SUBAPPLICATION SRV_SERVER (* ROS 2 SRV Server *)
  (* Standard: 61499-2 *)
  (* Version 1.0, 2023-03-14, derPi *)
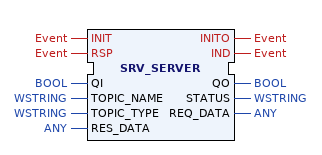
  EVENT_INPUT
    INIT; (* Initialization Request *)
    RSP; (* Application Response to IND *)
  END_EVENT
  EVENT_OUTPUT
    INITO; (* Initialization Confirm *)
    IND; (* Confirmation of Requested Service *)
  END_EVENT
  VAR_INPUT
    QI : BOOL; (* Input Event Qualifier *)
    TOPIC_NAME : WSTRING; (* ROS 2 Topic Name *)
    TOPIC_TYPE : WSTRING; (* ROS 2 Topic Type *)
    RES_DATA : ANY; (* Response Data *)
  END_VAR
  VAR_OUTPUT
    QO : BOOL; (* Output Event Qualifier *)
    STATUS : WSTRING; (* Service Status *)
    REQ_DATA : ANY; (* Request Data *)
  END_VAR
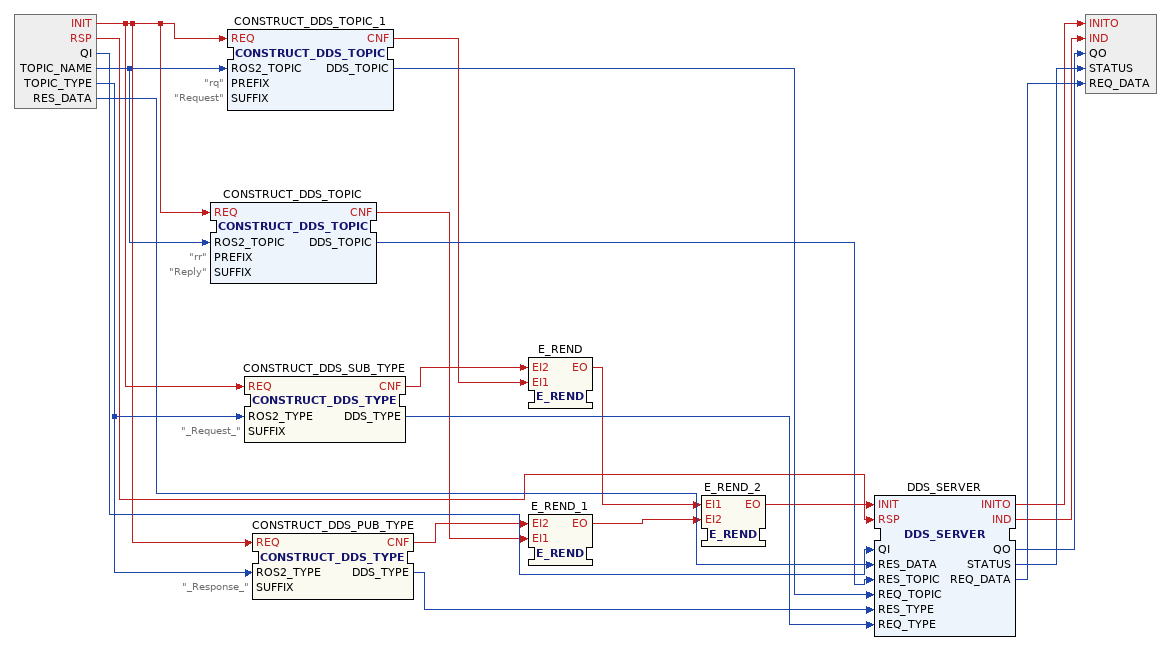
  FBS
    CONSTRUCT_DDS_SUB_TYPE : CONSTRUCT_DDS_TYPE(SUFFIX := "_Request_");
    CONSTRUCT_DDS_PUB_TYPE : CONSTRUCT_DDS_TYPE(SUFFIX := "_Response_");
    E_REND : E_REND;
    E_REND_1 : E_REND;
    E_REND_2 : E_REND;
  END_FBS
  SUBAPPS
    CONSTRUCT_DDS_TOPIC : CONSTRUCT_DDS_TOPIC(PREFIX := "rr", SUFFIX := "Reply");
    CONSTRUCT_DDS_TOPIC_1 : CONSTRUCT_DDS_TOPIC(PREFIX := "rq", SUFFIX := "Request");
    DDS_SERVER : DDS_SERVER;
  END_SUBAPPS
  EVENT_CONNECTIONS
    CONSTRUCT_DDS_SUB_TYPE.CNF TO E_REND.EI2;
    CONSTRUCT_DDS_PUB_TYPE.CNF TO E_REND_1.EI2;
    INIT TO CONSTRUCT_DDS_SUB_TYPE.REQ;
    INIT TO CONSTRUCT_DDS_PUB_TYPE.REQ;
    E_REND.EO TO E_REND_2.EI1;
    E_REND_1.EO TO E_REND_2.EI2;
    CONSTRUCT_DDS_TOPIC.CNF TO E_REND_1.EI1;
    INIT TO CONSTRUCT_DDS_TOPIC.REQ;
    CONSTRUCT_DDS_TOPIC_1.CNF TO E_REND.EI1;
    INIT TO CONSTRUCT_DDS_TOPIC_1.REQ;
    E_REND_2.EO TO DDS_SERVER.INIT;
    RSP TO DDS_SERVER.RSP;
    DDS_SERVER.INITO TO INITO;
    DDS_SERVER.IND TO IND;
  END_CONNECTIONS
  DATA_CONNECTIONS
    TOPIC_TYPE TO CONSTRUCT_DDS_SUB_TYPE.ROS2_TYPE;
    TOPIC_TYPE TO CONSTRUCT_DDS_PUB_TYPE.ROS2_TYPE;
    TOPIC_NAME TO CONSTRUCT_DDS_TOPIC.ROS2_TOPIC;
    TOPIC_NAME TO CONSTRUCT_DDS_TOPIC_1.ROS2_TOPIC;
    QI TO DDS_SERVER.QI;
    DDS_SERVER.QO TO QO;
    DDS_SERVER.STATUS TO STATUS;
    DDS_SERVER.REQ_DATA TO REQ_DATA;
    RES_DATA TO DDS_SERVER.RES_DATA;
    CONSTRUCT_DDS_TOPIC.DDS_TOPIC TO DDS_SERVER.RES_TOPIC;
    CONSTRUCT_DDS_TOPIC_1.DDS_TOPIC TO DDS_SERVER.REQ_TOPIC;
    CONSTRUCT_DDS_PUB_TYPE.DDS_TYPE TO DDS_SERVER.RES_TYPE;
    CONSTRUCT_DDS_SUB_TYPE.DDS_TYPE TO DDS_SERVER.REQ_TYPE;
  END_CONNECTIONS
END_SUBAPPLICATION
